TYPE hmiCommandsSmallPosCorrection_TypeStruct :
STRUCT
	
	positionCorrection	: REAL;
	execute				: BOOL;

END_STRUCT
END_TYPE

(* stored: Version 1.1.0.1
   DUT hmiCommandsSmallPosCorrection_TypeStruct: Id {72725890-5698-488e-826b-958ce06b38de} *)
